TYPE HardWareIO :
STRUCT
	HWInput			:HardwareInput;
	HWOutput		:HardwareOutput;
END_STRUCT
END_TYPE

(* stored: Version 1.1.0.1, ProductVersion 3.1.4022.16
   DUT HardWareIO: Id {bbd1e568-8a60-4eb5-adf1-50e10b8ad1b7} *)
